FUNCTION_BLOCK S1SkipS2 (* Basic Function Block Type *)
  (* Standard: 61499-2 *)
  (* Version 0.0, 7/5/2026, Schneider Electric, Template *)
  PACKAGE SE.Nereda;
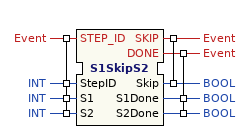
  EVENT_INPUT
    STEP_ID WITH StepID, S1, S2;
  END_EVENT
  EVENT_OUTPUT
    SKIP WITH Skip;
    DONE WITH S1Done, S2Done;
  END_EVENT
  VAR_INPUT
    StepID : INT;
    S1 : INT;
    S2 : INT;
  END_VAR
  VAR_OUTPUT
    Skip : BOOL;
    S1Done : BOOL;
    S2Done : BOOL;
  END_VAR
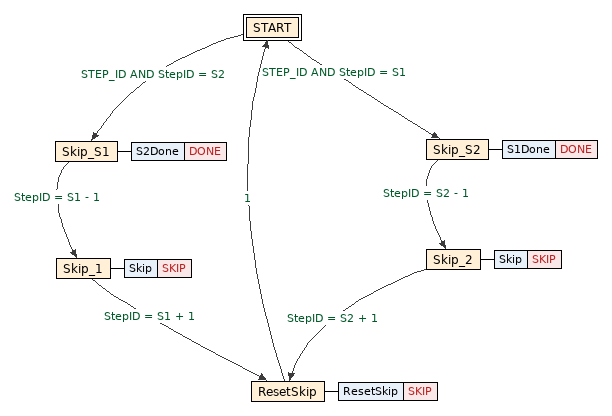
  EC_STATES
    START; (* Initial State *)
    Skip_S1 : S2Done -> DONE;
    Skip_S2 : S1Done -> DONE;
    Skip_1 : Skip -> SKIP;
    ResetSkip : ResetSkip -> SKIP;
    Skip_2 : Skip -> SKIP;
  END_STATES
  EC_TRANSITIONS
    START TO Skip_S1 := STEP_ID AND StepID = S2;
    Skip_S1 TO Skip_1 := StepID = S1 - 1;
    Skip_1 TO ResetSkip := StepID = S1 + 1;
    ResetSkip TO START := 1;
    START TO Skip_S2 := STEP_ID AND StepID = S1;
    Skip_S2 TO Skip_2 := StepID = S2 - 1;
    Skip_2 TO ResetSkip := StepID = S2 + 1;
  END_TRANSITIONS
  ALGORITHM Skip IN ST:
;
Skip := TRUE;
  END_ALGORITHM
  ALGORITHM ResetSkip IN ST:
;
Skip := FALSE;
  END_ALGORITHM
  ALGORITHM S2Done IN ST:
;
S1Done := FALSE;
S2Done := TRUE;
  END_ALGORITHM
  ALGORITHM S1Done IN ST:
;
S1Done := TRUE;
S2Done := FALSE;
  END_ALGORITHM
END_FUNCTION_BLOCK
